// TIA Portal V20 export
FUNCTION_BLOCK "FB_Fixture"   // FB37, SCL
{ S7_Optimized_Access := 'TRUE' }
// stored: MemoryReserve 100, SetENOAutomatically false
   VAR_INPUT
      iOpenCtrl { ExternalAccessible := 'False'; ExternalVisible := 'False'; ExternalWritable := 'False'} : Bool;
      iCloseCtrl { ExternalAccessible := 'False'; ExternalVisible := 'False'; ExternalWritable := 'False'} : Bool;
      iHoldReq : Bool;   // Hold Request
      iVacuumReq : Bool;   // Vacuum Request
      iBlowingReq : Bool;   // Blowing Request
      iMonitorTime : Time;
   END_VAR
   VAR_OUTPUT
      oClampOpening : Bool;   // Clamp Opening
      oClampClosing : Bool;   // Clamp Closing
      oVacuumActivation : Bool;   // Vacuum Activation
      oBlowingActivation : Bool;   // Blowing Activation
      oErrorCode { ExternalAccessible := 'False'; ExternalVisible := 'False'; ExternalWritable := 'False'} : Int;
   END_VAR
   VAR
      sMonitorTimer : TON_TIME;
   END_VAR
BEGIN
   REGION Description header 
       //==================================================================================
       // POSALUX Swiss SA / (C) Copyright 2025
       //----------------------------------------------------------------------------------
       // Title: FB_Fixture
       // Comment/Function: 
       // Author: Fabien WALDT
       // Engineering: TIA Portal v17
       //----------------------------------------------------------------------------------
       // Change log table:
       // Version  | Date     | Expert in charge | Changes applied
       // ---------|----------|------------------|-----------------------------------------
       // 00.00.01 | 20250502 | WFA              | First released version
       // =================================================================================
   END_REGION

   REGION Init
   // Outputs Initialisation
   #oClampOpening := FALSE;
   #oClampClosing := FALSE;
   #oVacuumActivation := FALSE;
   #oBlowingActivation := FALSE;
   END_REGION

   REGION Clamp Opening - Closing
       IF #iHoldReq AND NOT "DB_MachineOptions".Fixture.Passive_Open THEN
           #oClampOpening := FALSE;
           #oClampClosing := TRUE;
       ELSIF NOT #iHoldReq AND NOT "DB_MachineOptions".Fixture.Passive_Open THEN
           #oClampOpening := TRUE;
           #oClampClosing := FALSE;
       END_IF;
   END_REGION

   REGION Vacuum Activation
       #oVacuumActivation := #iVacuumReq;
   END_REGION

   REGION Blowing Activation
       #oBlowingActivation := #iBlowingReq;
   END_REGION

   REGION Monitoring Timer
       #sMonitorTimer(IN := (#oClampOpening AND NOT #iOpenCtrl) 
                         OR (#oClampClosing AND NOT #iCloseCtrl)
                         OR (NOT #iOpenCtrl AND NOT #iCloseCtrl)
                         OR (#iOpenCtrl AND #iCloseCtrl),
                                PT := #iMonitorTime);
   END_REGION

   REGION Error Codes
       #oErrorCode := 0;        // Code 0: No Error
       IF #oClampOpening AND #sMonitorTimer.Q THEN
           #oErrorCode := 1;    // Code 1: Error Open Command Plus
       ELSIF #oClampClosing AND #sMonitorTimer.Q THEN
           #oErrorCode := 2;    // Code 2: Error Close Command Minus
       ELSIF NOT #iOpenCtrl AND NOT #iOpenCtrl AND #sMonitorTimer.Q THEN
           #oErrorCode := 3;    // Code 3: Error Timeout Position OFF   
       ELSIF #iOpenCtrl AND #iOpenCtrl AND #sMonitorTimer.Q THEN
           #oErrorCode := 4;    // Code 4: Error Timeout Position ON       
       END_IF;
   END_REGION
END_FUNCTION_BLOCK
